{attribute 'linkalways'} 
{attribute 'no_explicit_call' := 'This FB is a CLASS and must be accessed using methods or properties'}
{attribute 'enable_dynamic_creation'}
FUNCTION_BLOCK _ETcVnEstimationAlgorithm EXTENDS EnumDatatypeBase
VAR
	localData : ETcVnEstimationAlgorithm;
	activeData : REFERENCE TO ETcVnEstimationAlgorithm;
	enumBaseDatatype : _DINT(localData);
END_VAR

METHOD PRIVATE AddLocalEnumeration
VAR_INPUT
	Enumeration : T_MAXSTRING;
	Value : ETcVnEstimationAlgorithm;
END_VAR
AddEnumeration(Enumeration, Value);
END_METHOD

PROPERTY PUBLIC Address : PVOID
GET
Address := ADR(activeData);
END_GET
END_PROPERTY

METHOD PUBLIC ClearReference
VAR_INPUT
END_VAR
activeData REF= localData;
SetBaseDatatypeReference();
END_METHOD

METHOD PUBLIC Clone : I_Datatype
VAR
    pClone : POINTER TO _ETcVnEstimationAlgorithm;
END_VAR
pClone := __NEW(_ETcVnEstimationAlgorithm(InitialValue := Value));
Clone := pClone^;
END_METHOD

METHOD FB_init : BOOL
VAR_INPUT
	bInitRetains : BOOL; // if TRUE, the retain variables are initialized (warm start / cold start)
	bInCopyCode : BOOL;  // if TRUE, the instance afterwards gets moved into the copy code (online change)
	InitialValue : ETcVnEstimationAlgorithm;
END_VAR
localData := InitialValue;
AddBaseDatatype(enumBaseDatatype);
ClearReference();

AddLocalEnumeration('TCVN_EA_DEFAULT', ETcVnEstimationAlgorithm.TCVN_EA_DEFAULT);
AddLocalEnumeration('TCVN_EA_LMEDS', ETcVnEstimationAlgorithm.TCVN_EA_LMEDS);
AddLocalEnumeration('TCVN_EA_RANSAC', ETcVnEstimationAlgorithm.TCVN_EA_RANSAC);
AddLocalEnumeration('TCVN_EA_RHO', ETcVnEstimationAlgorithm.TCVN_EA_RHO);
END_METHOD

PROPERTY PUBLIC Identifier : T_MAXSTRING
GET
Identifier := 'ETcVnEstimationAlgorithm';
END_GET
END_PROPERTY

METHOD IsEnumeratorValueEqual : BOOL
VAR_INPUT
	Enumerator : I_KeyValueForwardEnumerator;
END_VAR
VAR
	storedValue : ETcVnEstimationAlgorithm;
END_VAR
IF NOT Enumerator.TryGet(storedValue) THEN
	RETURN;
END_IF

IsEnumeratorValueEqual := storedValue = activeData;
END_METHOD

METHOD PUBLIC MakeReferenceTo
VAR_INPUT
	ReferenceTarget : REFERENCE TO ETcVnEstimationAlgorithm;
END_VAR
activeData REF= ReferenceTarget;
SetBaseDatatypeReference();
END_METHOD

METHOD PROTECTED SetBaseDatatypeReference
VAR_INPUT
END_VAR
enumBaseDatatype.MakeReferenceTo(activeData);
END_METHOD

PROPERTY PUBLIC Size : UDINT
GET
Size := SIZEOF(activeData);
END_GET
END_PROPERTY

METHOD TryMakeReferenceTo : BOOL
VAR_INPUT
	Target : I_Datatype;
END_VAR
VAR
	targetAsEnum : I_EnumDatatype;
	pTargetData : POINTER TO ETcVnEstimationAlgorithm;
END_VAR
IF NOT Target.TryResolveAsEnumDatatype(targetAsEnum) THEN
	RETURN;
END_IF

IF targetAsEnum.Identifier <> Identifier THEN
	RETURN;
END_IF

pTargetData := Target.Address;
activeData REF= pTargetData^;
SetBaseDatatypeReference();
TryMakeReferenceTo := TRUE;
END_METHOD

PROPERTY PUBLIC Value : ETcVnEstimationAlgorithm
GET
Value := activeData;
END_GET
SET
activeData := Value;
END_SET
END_PROPERTY

END_FUNCTION_BLOCK

(* stored: Version 1.1.0.1
   POU _ETcVnEstimationAlgorithm: Id {c493b84e-1988-44f5-bf66-1448d75e0045}, SpecialFunc None
   Folder Constructor: Id {48becb62-8a38-47dd-bff4-7a7326183ee1}
   Folder Private: Id {8d9b2738-0d1e-42dd-9b7a-9f7528b7bfcb}
   Folder Protected: Id {1205a05f-a5f5-4172-ad40-33394436872f}
   Method AddLocalEnumeration: Id {a5434fc5-58fb-472a-b1e5-fbfe8452ab51}
   Property Address: Id {af7f00cf-8ed1-42ff-b187-46fd299e6513}
   Get Get: Id {cf3c9819-6e0f-4dba-a688-9878ae917c3b}
   Method ClearReference: Id {8a6d0d23-0bd8-499d-a75a-b1a4c898b252}
   Method Clone: Id {79a4544f-826b-4137-ae0a-08b2e2a2a6b5}
   Method FB_init: Id {ba732033-7426-4905-90f5-8972fc4a8a96}
   Property Identifier: Id {7c117e14-af71-4f01-ab10-a7f9d67049af}
   Get Get: Id {6d264a4c-a6f5-40f2-ba11-1aaa9f1dfd2b}
   Method IsEnumeratorValueEqual: Id {c0441bdb-88ea-4ab6-964c-85c176061e9e}
   Method MakeReferenceTo: Id {14084309-7bab-43cc-a351-d9ce8eab4d32}
   Method SetBaseDatatypeReference: Id {5083d5b9-af91-4e55-a890-cb443019a7e7}
   Property Size: Id {9a9bcc17-e269-4a35-97f2-36ff7f86d7fe}
   Get Get: Id {8904d15e-5c67-4f3e-b54a-e39f601b47c0}
   Method TryMakeReferenceTo: Id {b0a0653a-4674-4ea9-b9f0-f1f328be96a3}
   Property Value: Id {e2a9d8ca-49b1-429a-bc7f-e2b5a2c51b15}
   Get Get: Id {8eade530-97ca-411c-af63-2940e1b7fbbf}
   Set Set: Id {2b0961e3-2114-4dda-a3ec-504a3a5669b0} *)
